(**************************************************************************************
 * 	Application		:	BoxControl Framework
 *	Revision		:	$Revision: 404529 $
 *	Revision date	:	$Date: 2018-04-23 08:21:38 +0200 (Mo., 23 Apr 2018) $
 *	Last changed by	:	$Author: b7bolm $
 *	URL				:	$URL: http://almscdc.swisslog.com/repo/SWPD/Development/BoxControlFramework/20_Release/trunk/01_Software/BCF/BCF/JumpStart/20_Product/10_App/10_Base/10_Lib/00_GVLs/SDO_Table.TcGVL $
 *
 *	Purpose			:	SDO signals - Separated due to debug reasons.
 *
 * ------------------------------------------------------------------------------------
 *	Copyright Swisslog [IP AG], Switzerland. All rights reserved.
 * 
 * ------------------------------------------------------------------------------------
 *	
 * 	Revision History: 
 *
 * 	VERSION			DATE			INITIALS			DESCRIPTION
 *	0.1				01.01.2001		swl					Example
 *
 **************************************************************************************)

VAR_GLOBAL CONSTANT
	NUMBER_OF_SDO_SIGNALS			: INT := 9999; // Number of SDO signals, max 9999 
END_VAR
 
VAR_GLOBAL
	SDOSignalNumber					: ARRAY [0..NUMBER_OF_SDO_SIGNALS] OF BOOL; // SDO table
END_VAR

(* stored: Version 1.1.0.1, ProductVersion 3.1.4022.12
   GVL SDO_Table: Id {e300bd8c-2a22-4217-9354-b30e085f3ef5} *)
